// Exemple illustrates how to write a (XBA) schedulers 'object property reference' property (BACnet).
FUNCTION_BLOCK FB_BACnet_ObjPropRef EXTENDS FB_BA_View
VAR
	bWrite			: BOOL;
	
	MySched			: FB_BA_SchedM := (
						iParent					:= THIS^,
						sDescription			:= '{Some schedule}',
						aStateText				:= [ 'Aus', 'Stufe 1', 'Stufe 2' ]
					);
END_VAR

SUPER^();

MySched();

IF (bWrite) THEN
	bWrite := FALSE;
	
	WriteReference(F_BACnet_GetObjId(E_BACnetObjType.ObjMultiStateValue, 12345), E_BACnetPropIdentifier.PropPresentValue);
//	[Alternative]
//	WriteReferenceRm(F_BACnet_GetObjId(E_BACnetObjType.ObjMultiStateValue, 12345), 1000, E_BACnetPropIdentifier.PropPresentValue);
END_IF

// Write reference to a local BACnet object.
METHOD WriteReference : BOOL
VAR_INPUT
	tObjectID		: T_BACnet_ObjectIdentifier		:= 16#FFFFFFFF;
	eProperty		: E_BACnetPropIdentifier		:= E_BACnetPropIdentifier.PropPresentValue;
END_VAR
WriteReference := WriteReferenceRm(tObjectID, 16#FFFFFFFF, eProperty);
END_METHOD

// Write reference to a remote BACnet object.
METHOD WriteReferenceRm : BOOL
VAR_INPUT
	tObjectID		: T_BACnet_ObjectIdentifier		:= 16#FFFFFFFF;
	nDeviceID		: UDINT							:= 16#FFFFFFFF;
	eProperty		: E_BACnetPropIdentifier		:= E_BACnetPropIdentifier.PropPresentValue;
END_VAR
VAR
	stRef			: ST_BACnet_ObjectPropertyReference := (
						tObjectID		:= tObjectID,
						nDeviceID		:= nDeviceID,
						ePropertyId		:= eProperty
					);
END_VAR
VAR
	_iObj			: I_BA_Object;
	_fbBACnetObj	: POINTER TO FB_BACnet_BaseObject;
	_hRes			: HRESULT;
END_VAR
// Receive internal BACnet object from BA object:
IF (NOT MySched.GetBACnetObject(fbObject=>_fbBACnetObj)) THEN
	MySched.LogMsg.Show(ADSLOG_MSGTYPE_ERROR, 'OPR10', 'Failed to receive internal BACnet object!', TRUE);
ELSE
	// Write property:
	WriteReferenceRm := SUCCEEDED(_fbBACnetObj^.WritePropertyReferenceList1x(E_BACnetPropIdentifier.PropListOfObjectPropertyReferences, stRef));
END_IF
END_METHOD

END_FUNCTION_BLOCK

(* stored: Version 1.1.0.1, ProductVersion 3.1.4024.12
   POU FB_BACnet_ObjPropRef: Id {deb3c8ae-6758-45b6-9557-fb2097912fea}, SpecialFunc None
   Method WriteReference: Id {97f3dbd8-1654-408a-8f8a-57768a421f0f}
   Method WriteReferenceRm: Id {d8fdb4f2-1ed2-44ad-a901-1866a61228a6} *)
